// TIA Portal project "Vessel" (V12)

(* hardware
DEVICE "S7-1200 station_1"  SIMATIC 1200-Station
   slot 0: "S7-1200 rack"  Rack  V1.0
   slot 1: "PLC_1"  CPU 1212C DC/DC/DC  6ES7 212-1AD30-0XB0  V2.2
   slot 2: "AI4 x 13 bits / AQ2 x 14 bits_2"  6ES7 234-4HE32-0XB0  V2.0
*)

// ===== PLC "PLC_1"  CPU 1212C DC/DC/DC =====

VAR_GLOBAL   // PLC tag table "Default tag table"
   "PH_Sensor_AI" AT %IW112 : Word;
   "Tempreture_Sensor_AI" AT %IW114 : Word;
   "Mixer_Speed_AO" AT %QW112 : Word;
   "PH_Sensor" AT %MW2 : Word;
   "Tempreture_Sensor" AT %MW4 : Word;
   "Mixer_Speed" AT %MW6 : Word;
   "Valve1_DO" AT %Q0.0 : Bool;
   "Valve2_DO" AT %Q0.1 : Bool;
   "Valve3_DO" AT %Q0.2 : Bool;
   "Valve4_DO" AT %Q0.3 : Bool;
   "Valve5_DO" AT %Q0.4 : Bool;
   "Valve1" AT %M1.0 : Bool;
   "Valve2" AT %M1.1 : Bool;
   "Valve3" AT %M1.2 : Bool;
   "Valve4" AT %M1.3 : Bool;
   "Valve5" AT %M1.4 : Bool;
   "Mixer_DO" AT %Q0.5 : Bool;
   "Mixer" AT %M1.5 : Bool;
END_VAR

FUNCTION "Scale" : Void   // FC1, LAD
{ S7_Optimized_Access := 'FALSE' }
VERSION : 0.1
   VAR_TEMP
      temp_ph : Real;
      temp_tempreture : Real;
      temp_speed : Real;
   END_VAR
BEGIN

REGION Network 1
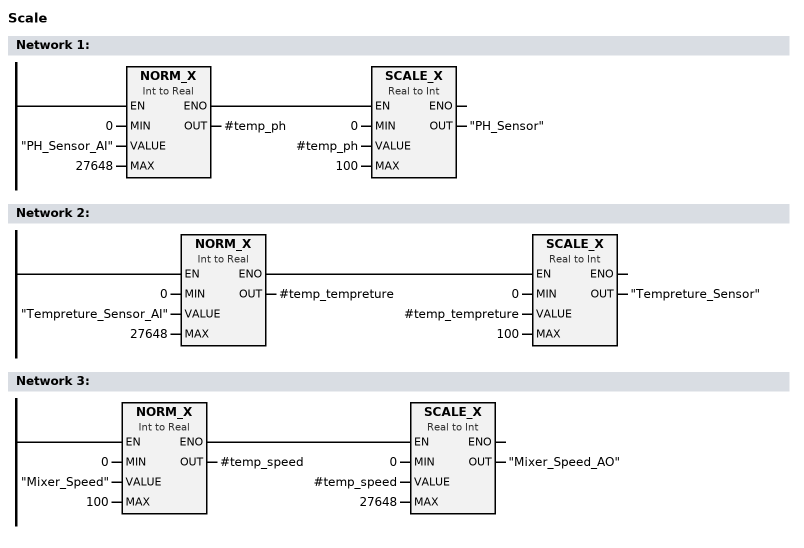
   RUNG wire#powerrail
      { S7_Templates := "[SrcType := Int, DestType := Real]"; S7_GenerateENO := "TRUE" } Normalize(min := 0, value := "PH_Sensor_AI", max := 27648, out => #temp_ph)
      { S7_Templates := "[SrcType := Real, DestType := Int]"; S7_GenerateENO := "TRUE" } Scale(min := 0, value := #temp_ph, max := 100, out => "PH_Sensor")
   END_RUNG
   // the same network as SCL:
   // ENO of a box is taken as its EN; it also drops when the box reports an error
   #temp_ph := NORM_X(MIN := 0, VALUE := "PH_Sensor_AI", MAX := 27648);
   "PH_Sensor" := SCALE_X(MIN := 0, VALUE := #temp_ph, MAX := 100);
END_REGION

REGION Network 2
   RUNG wire#powerrail
      { S7_Templates := "[SrcType := Int, DestType := Real]"; S7_GenerateENO := "TRUE" } Normalize(min := 0, value := "Tempreture_Sensor_AI", max := 27648, out => #temp_tempreture)
      { S7_Templates := "[SrcType := Real, DestType := Int]"; S7_GenerateENO := "TRUE" } Scale(min := 0, value := #temp_tempreture, max := 100, out => "Tempreture_Sensor")
   END_RUNG
   // the same network as SCL:
   // ENO of a box is taken as its EN; it also drops when the box reports an error
   #temp_tempreture := NORM_X(MIN := 0, VALUE := "Tempreture_Sensor_AI", MAX := 27648);
   "Tempreture_Sensor" := SCALE_X(MIN := 0, VALUE := #temp_tempreture, MAX := 100);
END_REGION

REGION Network 3
   RUNG wire#powerrail
      { S7_Templates := "[SrcType := Int, DestType := Real]"; S7_GenerateENO := "TRUE" } Normalize(min := 0, value := "Mixer_Speed", max := 100, out => #temp_speed)
      { S7_Templates := "[SrcType := Real, DestType := Int]"; S7_GenerateENO := "TRUE" } Scale(min := 0, value := #temp_speed, max := 27648, out => "Mixer_Speed_AO")
   END_RUNG
   // the same network as SCL:
   // ENO of a box is taken as its EN; it also drops when the box reports an error
   #temp_speed := NORM_X(MIN := 0, VALUE := "Mixer_Speed", MAX := 100);
   "Mixer_Speed_AO" := SCALE_X(MIN := 0, VALUE := #temp_speed, MAX := 27648);
END_REGION
END_FUNCTION

FUNCTION "Valves_Control" : Void   // FC2, LAD
{ S7_Optimized_Access := 'FALSE' }
VERSION : 0.1
BEGIN

REGION Network 2
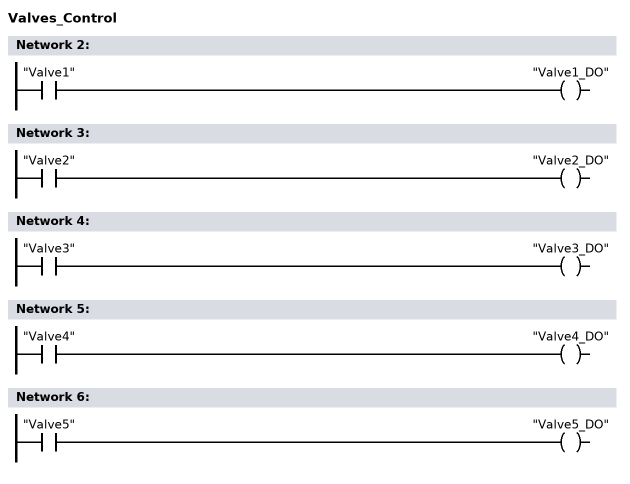
   RUNG wire#powerrail
      Contact( "Valve1" )
      Coil( "Valve1_DO" )
   END_RUNG
   // the same network as SCL:
   "Valve1_DO" := "Valve1";
END_REGION

REGION Network 3
   RUNG wire#powerrail
      Contact( "Valve2" )
      Coil( "Valve2_DO" )
   END_RUNG
   // the same network as SCL:
   "Valve2_DO" := "Valve2";
END_REGION

REGION Network 4
   RUNG wire#powerrail
      Contact( "Valve3" )
      Coil( "Valve3_DO" )
   END_RUNG
   // the same network as SCL:
   "Valve3_DO" := "Valve3";
END_REGION

REGION Network 5
   RUNG wire#powerrail
      Contact( "Valve4" )
      Coil( "Valve4_DO" )
   END_RUNG
   // the same network as SCL:
   "Valve4_DO" := "Valve4";
END_REGION

REGION Network 6
   RUNG wire#powerrail
      Contact( "Valve5" )
      Coil( "Valve5_DO" )
   END_RUNG
   // the same network as SCL:
   "Valve5_DO" := "Valve5";
END_REGION
END_FUNCTION

FUNCTION "Mixer_Control" : Void   // FC3, LAD
{ S7_Optimized_Access := 'FALSE' }
VERSION : 0.1
BEGIN

REGION Network 1
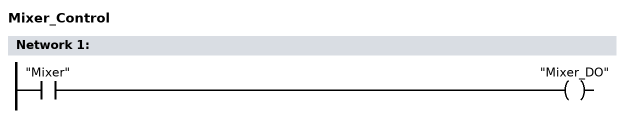
   RUNG wire#powerrail
      Contact( "Mixer" )
      Coil( "Mixer_DO" )
   END_RUNG
   // the same network as SCL:
   "Mixer_DO" := "Mixer";
END_REGION
END_FUNCTION

FUNCTION "Logging" : Void   // FC4, LAD
{ S7_Optimized_Access := 'FALSE' }
VERSION : 0.1
BEGIN

REGION Network 1
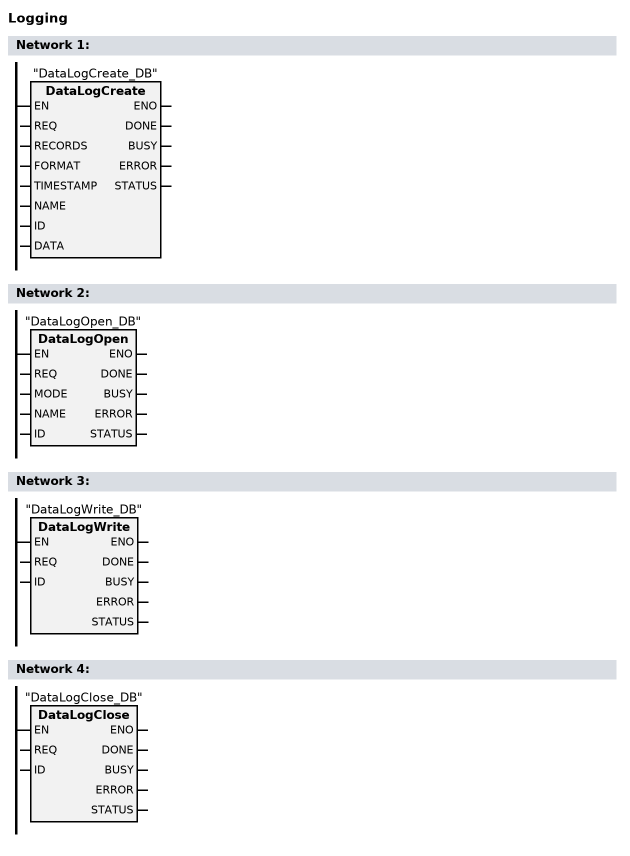
   "DataLogCreate_DB"();   // DataLogCreate
END_REGION

REGION Network 2
   "DataLogOpen_DB"();   // DataLogOpen
END_REGION

REGION Network 3
   "DataLogWrite_DB"();   // DataLogWrite
END_REGION

REGION Network 4
   "DataLogClose_DB"();   // DataLogClose
END_REGION
END_FUNCTION

ORGANIZATION_BLOCK "Main"   // OB1, LAD, ProgramCycle
TITLE = "Main Program Sweep (Cycle)"
{ S7_Optimized_Access := 'FALSE' }
VERSION : 0.1
BEGIN

REGION Network 1
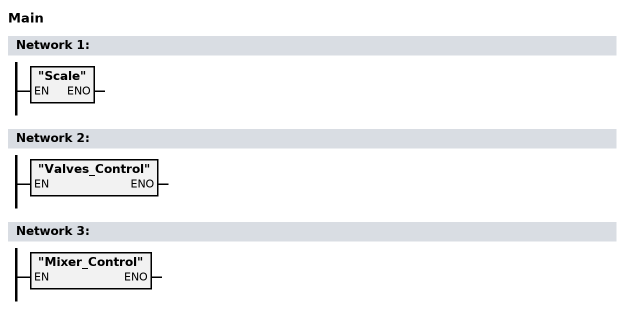
   RUNG wire#powerrail
      "Scale"()
   END_RUNG
   // the same network as SCL:
   "Scale"();
END_REGION

REGION Network 2
   RUNG wire#powerrail
      "Valves_Control"()
   END_RUNG
   // the same network as SCL:
   "Valves_Control"();
END_REGION

REGION Network 3
   RUNG wire#powerrail
      "Mixer_Control"()
   END_RUNG
   // the same network as SCL:
   "Mixer_Control"();
END_REGION
END_ORGANIZATION_BLOCK